// Mitsubishi GX Works2 project: PROJECT55   PLC: FX3G

// global labels: Global1
VAR_GLOBAL
  AnalogOutPut AT D8282 : INT;
  PacketReg AT D1100 : REAL;
  ChocolateToday AT D1102 : REAL;
  TotalChocolate AT D1110 : REAL;
  NutsToday AT D1104 : REAL;
  TotalNuts AT D1112 : REAL;
  FistokToday AT D1106 : REAL;
  TotalFistok AT D1114 : REAL;
  KadaifToday AT D1108 : REAL;
  TotalKadaif AT D1116 : REAL;
  InsertedValue AT M1 : BOOL;
  DayStarted AT M2 : BOOL;
  OutOfStock AT M3 : BOOL;
  DayEnded AT M4 : BOOL;
  EndDay AT X005 : BOOL;
  StartDay AT X007 : BOOL;
  WorkingLight AT Y007 : BOOL;
  MeltingStart AT X001 : BOOL;
END_VAR
VAR_GLOBAL CONSTANT
  MinChocolate : REAL := 400;
  MinNuts : REAL := 100;
  MinFistok : REAL := 120;
  MinKadaif : REAL := 60;
END_VAR
VAR_GLOBAL
  MeltingTank AT D1118 : REAL;
  TransferDone AT M7 : BOOL;
  Sense45 AT X002 : BOOL;
  MeltingLight AT Y001 : BOOL;
  MeltingDone AT M8 : BOOL;
  StockFinished AT M19 : BOOL;
  Sens4Molds AT X003 : BOOL;
  Molds AT D1120 : REAL;
  MoldsTransfer AT M9 : BOOL;
  InMolding AT TC1 : BOOL;
  MoldingFinished AT TS1 : BOOL;
  DuringMolding AT Y002 : BOOL;
END_VAR
VAR_GLOBAL CONSTANT
  MoldingTimee : INT := 40;
END_VAR
VAR_GLOBAL
  Sampling AT X004 : BOOL;
  AnalogInput1 AT D8280 : INT;
  ConvertAnalog AT D1200 : REAL;
END_VAR
VAR_GLOBAL CONSTANT
  ConertNum : REAL := 400;
END_VAR
VAR_GLOBAL
  UserChoice AT D1122 : REAL;
END_VAR
VAR_GLOBAL CONSTANT
  Min5 : REAL := 5;
END_VAR
VAR_GLOBAL
  MakeMixNuts AT M10 : BOOL;
  MakeDubai AT M11 : BOOL;
END_VAR
VAR_GLOBAL CONSTANT
  Count100 : REAL := 100;
END_VAR
VAR_GLOBAL
  MixNutsIngridiants AT M12 : BOOL;
END_VAR
VAR_GLOBAL CONSTANT
  Constant20 : REAL := 2;
  Constant120 : REAL := 2;
  Constant60 : REAL := 60;
END_VAR
VAR_GLOBAL
  DubaiIngridiants AT M13 : BOOL;
END_VAR
VAR_GLOBAL CONSTANT
  Constant100 : REAL := 1;
END_VAR
VAR_GLOBAL
  FillingTank AT D1124 : REAL;
  FillingMixNuts AT M14 : BOOL;
  FillingDubai AT M15 : BOOL;
  FillingDone AT M16 : BOOL;
  Blink AT M0 : BOOL;
  Blink3 AT TC2 : BOOL;
END_VAR
VAR_GLOBAL CONSTANT
  Constant5 : WORD := 5;
END_VAR
VAR_GLOBAL
  StopLight3 AT TS2 : BOOL;
  FillingLight1 AT Y003 : BOOL;
  Blink4 AT TC3 : BOOL;
  StopLight4 AT TS3 : BOOL;
  FillingLight2 AT Y004 : BOOL;
  BlinkingTimer AT TS4 : BOOL;
  StopBlinkingTimer AT TS4 : BOOL;
END_VAR
VAR_GLOBAL CONSTANT
  BlinkingTime : WORD := 50;
END_VAR
VAR_GLOBAL
  Cooling AT X006 : BOOL;
  CoolingTank AT D1126 : REAL;
  CoolingTransfer AT M17 : BOOL;
  CoolingTimer AT TC5 : BOOL;
  StopCoolingTimer AT TS5 : BOOL;
  CoolingLight AT Y006 : BOOL;
END_VAR
VAR_GLOBAL CONSTANT
  CoolingTime : INT := 30;
END_VAR
VAR_GLOBAL
  PackingMachine AT D1128 : REAL;
  PackingTransfer AT M18 : BOOL;
END_VAR
VAR_GLOBAL CONSTANT
  Packing : WORD := 4;
END_VAR
VAR_GLOBAL
  OnePack AT X000 : BOOL;
  PacketsCounter AT CC1 : BOOL;
  StopPacketsCounter AT CS1 : BOOL;
  PackingLight AT Y005 : BOOL;
END_VAR
VAR_GLOBAL CONSTANT
  Constant1 : REAL := 1;
  Constant40 : REAL := 40;
END_VAR
VAR_GLOBAL
  DailyPackets AT D1130 : REAL;
  Cooling1 AT M30 : BOOL;
END_VAR
VAR_GLOBAL CONSTANT
  Min6 : REAL := 6;
  Count20 : REAL := 20;
  Count120 : REAL := 120;
  Count60 : REAL := 60;
  Constant01 : WORD := 1;
END_VAR
VAR_GLOBAL
  PacketsRegg AT TS6 : BOOL;
  EndIteration AT M20 : BOOL;
  PacketsReg AT TS6 : BOOL;
END_VAR

// task Task_01 (event TRUE, interval 0, priority 31): POU_01

PROGRAM POU_01
(* structured ladder/FBD written out as ST: instructions are called as NAME(EN, inputs, outputs); _pN, _eN, _tN stand for wires *)
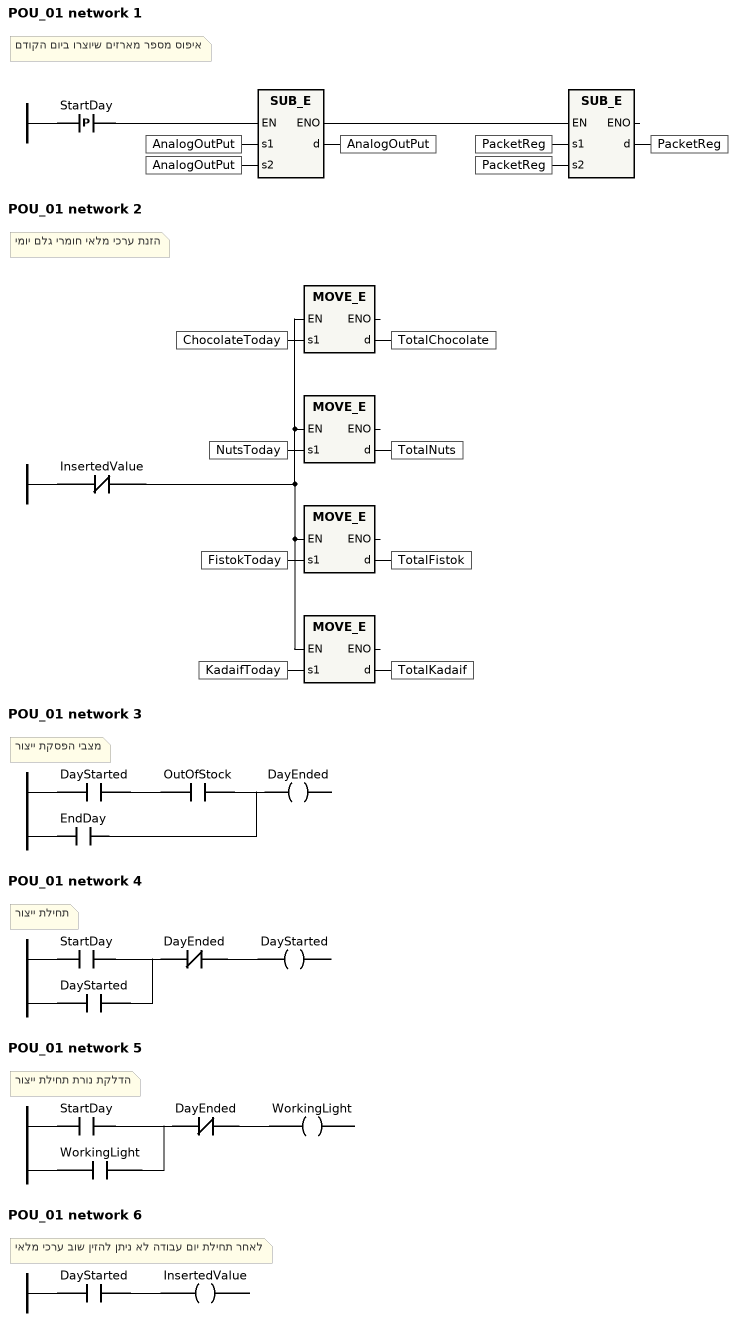
(* network 1 *)
(* איפוס מספר מארזים שיוצרו ביום הקודם *)
_e1 := SUB_E(LDP(TRUE, StartDay), AnalogOutPut, AnalogOutPut, AnalogOutPut);
SUB_E(_e1, PacketReg, PacketReg, PacketReg);
(* network 2 *)
(* הזנת ערכי מלאי חומרי גלם יומי *)
_p1 := NOT InsertedValue;
MOVE_E(_p1, ChocolateToday, TotalChocolate);
MOVE_E(_p1, NutsToday, TotalNuts);
MOVE_E(_p1, FistokToday, TotalFistok);
MOVE_E(_p1, KadaifToday, TotalKadaif);
(* network 3 *)
(* מצבי הפסקת ייצור *)
DayEnded := (DayStarted AND OutOfStock) OR EndDay;
(* network 4 *)
(* תחילת ייצור *)
DayStarted := (StartDay OR DayStarted) AND NOT DayEnded;
(* network 5 *)
(* הדלקת נורת תחילת ייצור *)
WorkingLight := (StartDay OR WorkingLight) AND NOT DayEnded;
(* network 6 *)
(* לאחר תחילת יום עבודה לא ניתן להזין שוב ערכי מלאי *)
InsertedValue := DayStarted;
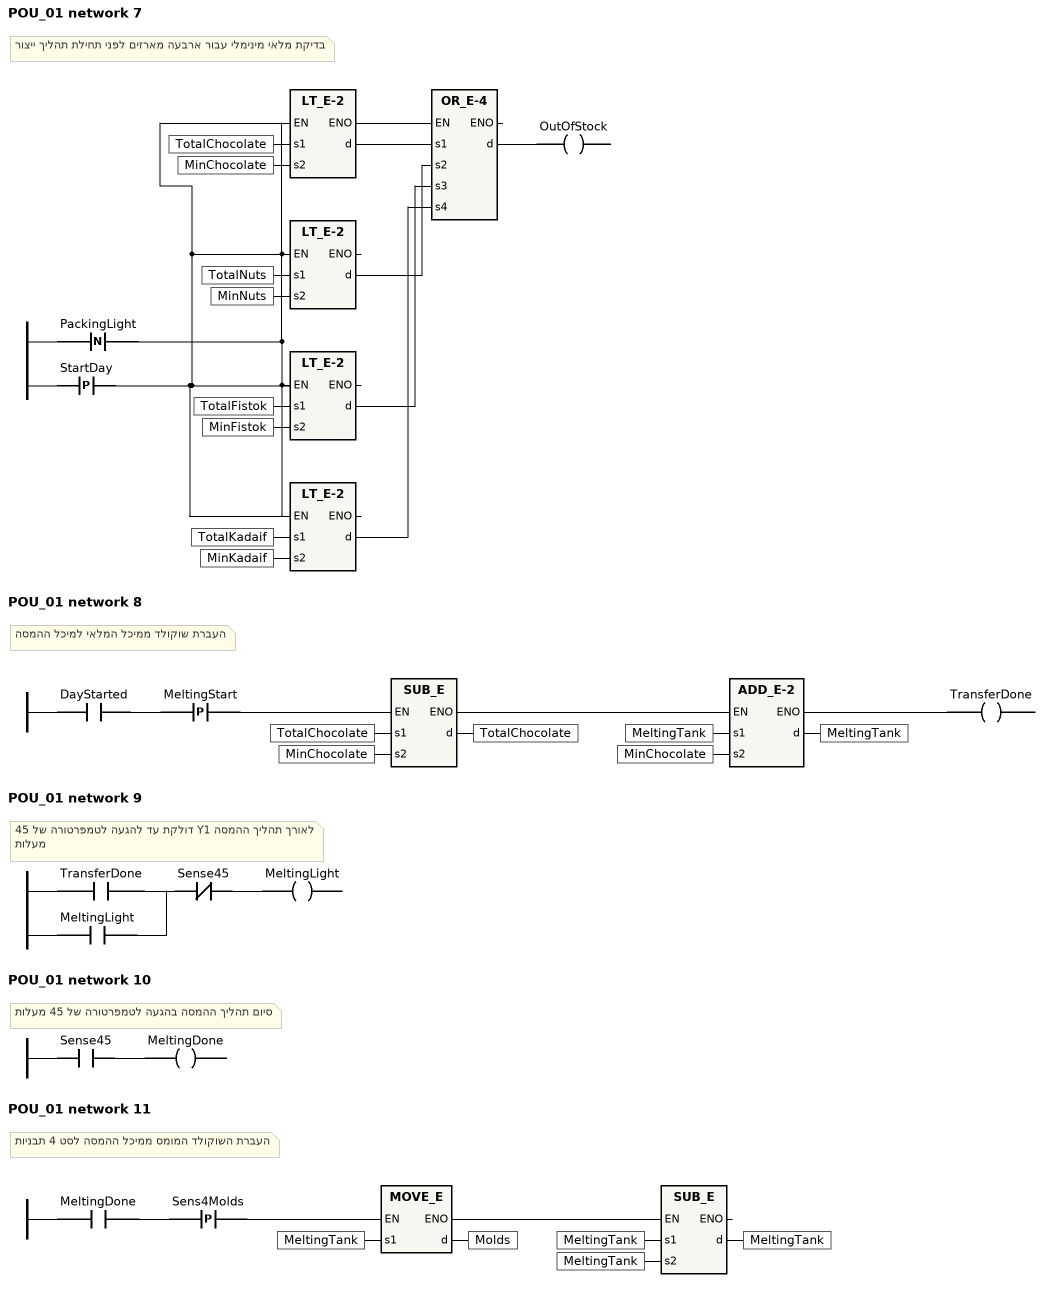
(* network 7 *)
(* בדיקת מלאי מינימלי עבור ארבעה מארזים לפני תחילת תהליך ייצור *)
_p1 := LDF(TRUE, PackingLight) OR LDP(TRUE, StartDay);
_e3 := LT_E(_p1, TotalChocolate, MinChocolate, _t2);
LT_E(_p1, TotalNuts, MinNuts, _t4);
LT_E(_p1, TotalFistok, MinFistok, _t5);
LT_E(_p1, TotalKadaif, MinKadaif, _t6);
OR_E(_e3, _t2, _t4, _t5, _t6, _t7);
OutOfStock := _t7;
(* network 8 *)
(* העברת שוקולד ממיכל המלאי למיכל ההמסה *)
_e1 := SUB_E(DayStarted AND LDP(TRUE, MeltingStart), TotalChocolate, MinChocolate, TotalChocolate);
_e2 := ADD_E(_e1, MeltingTank, MinChocolate, MeltingTank);
TransferDone := _e2;
(* network 9 *)
(* לאורך תהליך ההמסה Y1 דולקת עד להגעה לטמפרטורה של 45 מעלות *)
MeltingLight := (TransferDone OR MeltingLight) AND NOT Sense45;
(* network 10 *)
(* סיום תהליך ההמסה בהגעה לטמפרטורה של 45 מעלות *)
MeltingDone := Sense45;
(* network 11 *)
(* העברת השוקולד המומס ממיכל ההמסה לסט 4 תבניות *)
_e1 := MOVE_E(MeltingDone AND LDP(TRUE, Sens4Molds), MeltingTank, Molds);
SUB_E(_e1, MeltingTank, MeltingTank, MeltingTank);
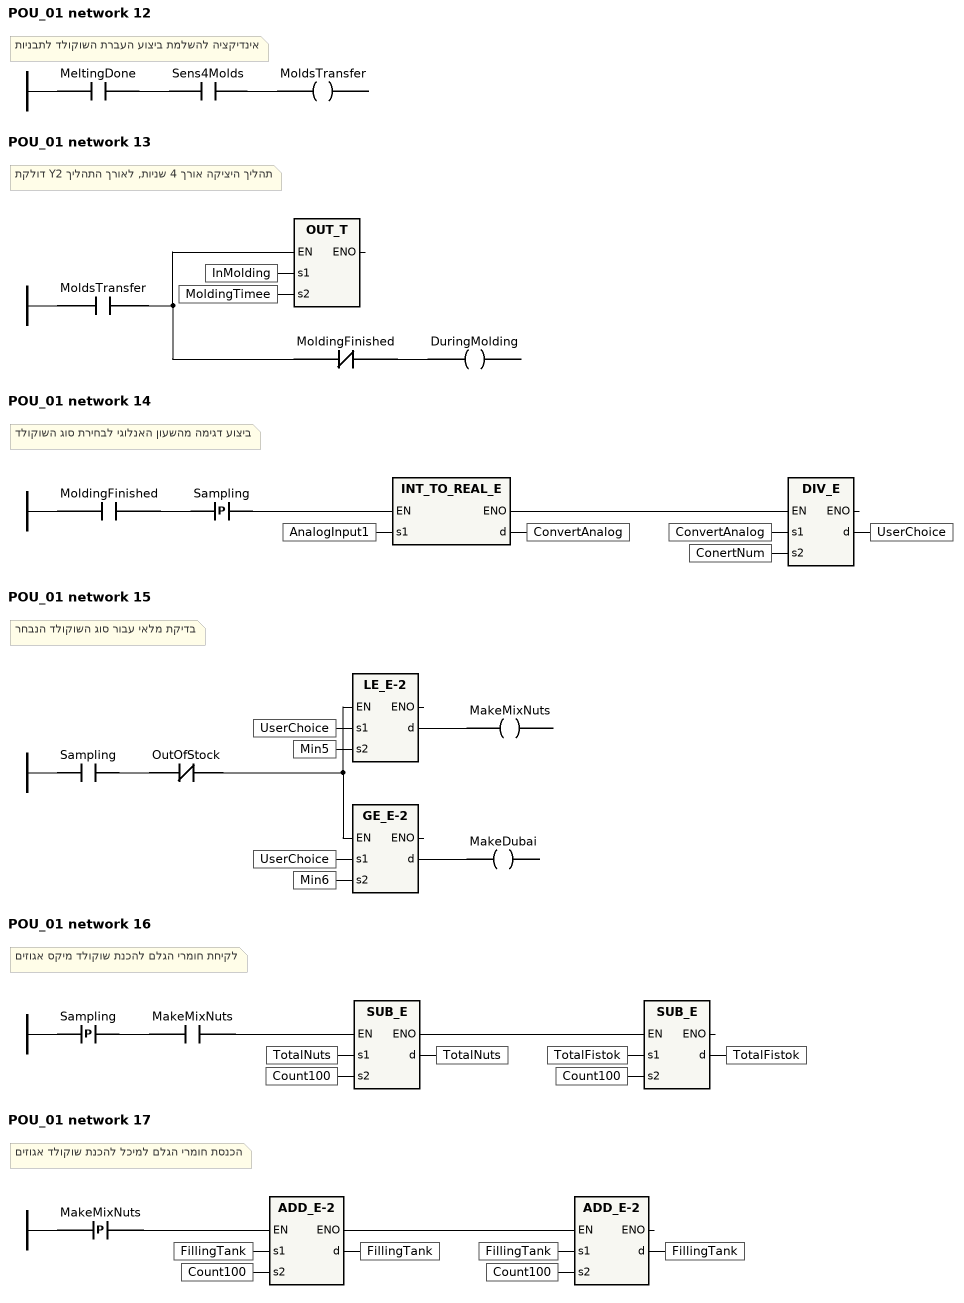
(* network 12 *)
(* אינדיקציה להשלמת ביצוע העברת השוקולד לתבניות *)
MoldsTransfer := MeltingDone AND Sens4Molds;
(* network 13 *)
(* תהליך היציקה אורך 4 שניות, לאורך התהליך Y2 דולקת *)
OUT_T(MoldsTransfer, InMolding, MoldingTimee);
DuringMolding := MoldsTransfer AND NOT MoldingFinished;
(* network 14 *)
(* ביצוע דגימה מהשעון האנלוגי לבחירת סוג השוקולד *)
_e1 := INT_TO_REAL_E(MoldingFinished AND LDP(TRUE, Sampling), AnalogInput1, ConvertAnalog);
DIV_E(_e1, ConvertAnalog, ConertNum, UserChoice);
(* network 15 *)
(* בדיקת מלאי עבור סוג השוקולד הנבחר *)
_p1 := Sampling AND NOT OutOfStock;
LE_E(_p1, UserChoice, Min5, _t2);
MakeMixNuts := _t2;
GE_E(_p1, UserChoice, Min6, _t3);
MakeDubai := _t3;
(* network 16 *)
(* לקיחת חומרי הגלם להכנת שוקולד מיקס אגוזים *)
_e1 := SUB_E(LDP(TRUE, Sampling) AND MakeMixNuts, TotalNuts, Count100, TotalNuts);
SUB_E(_e1, TotalFistok, Count100, TotalFistok);
(* network 17 *)
(* הכנסת חומרי הגלם למיכל להכנת שוקולד אגוזים *)
_e1 := ADD_E(LDP(TRUE, MakeMixNuts), FillingTank, Count100, FillingTank);
ADD_E(_e1, FillingTank, Count100, FillingTank);
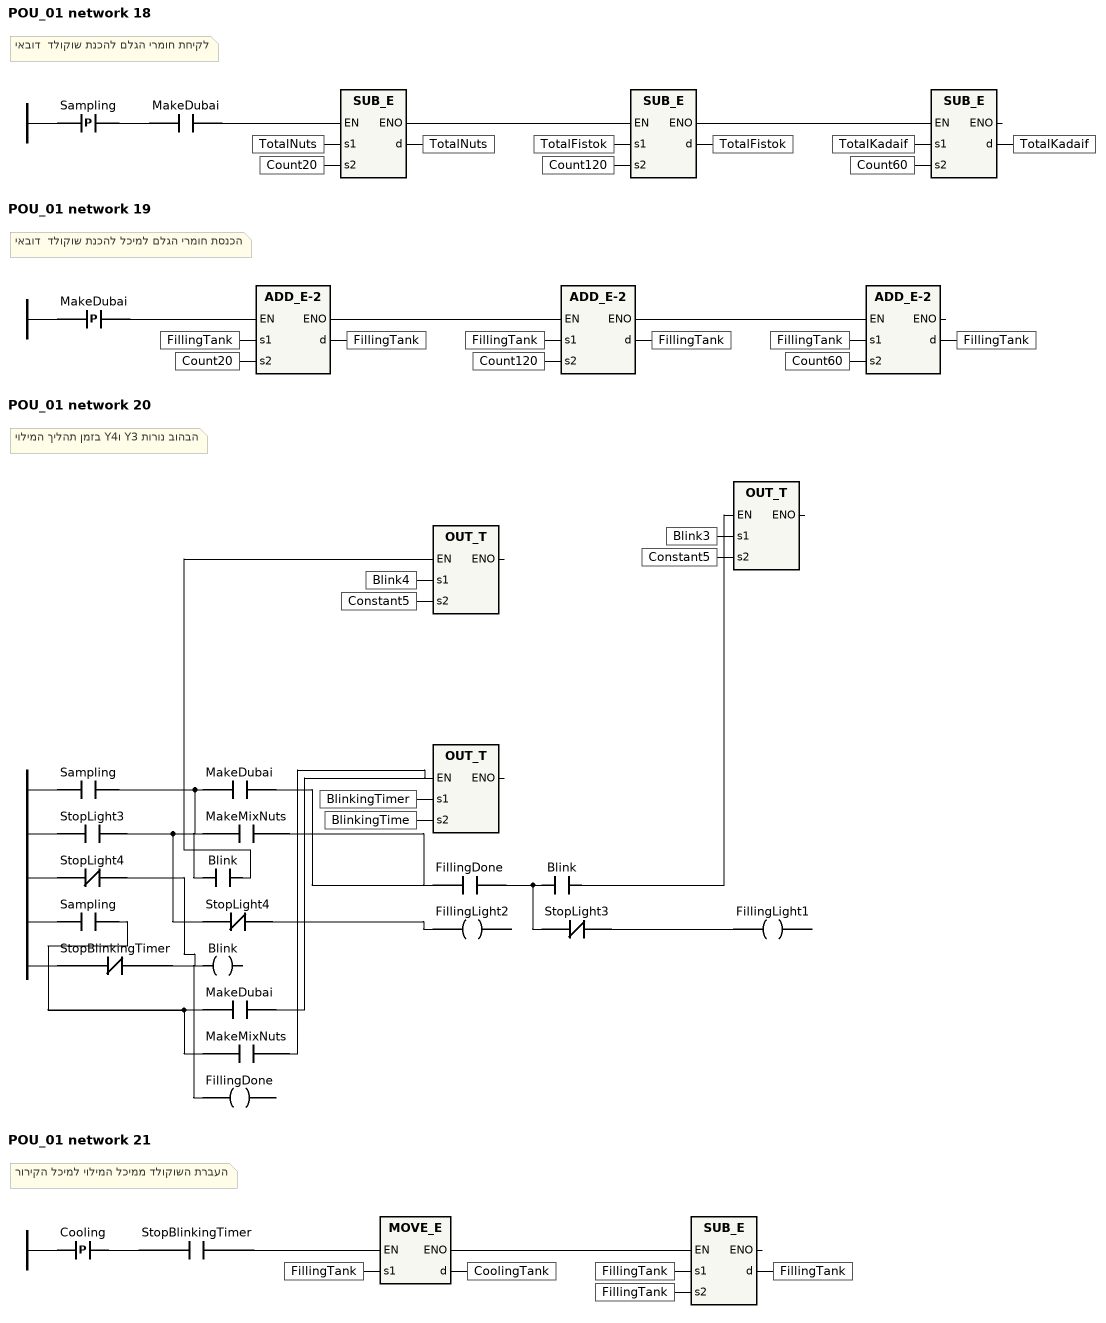
(* network 18 *)
(* לקיחת חומרי הגלם להכנת שוקולד  דובאי *)
_e1 := SUB_E(LDP(TRUE, Sampling) AND MakeDubai, TotalNuts, Count20, TotalNuts);
_e2 := SUB_E(_e1, TotalFistok, Count120, TotalFistok);
SUB_E(_e2, TotalKadaif, Count60, TotalKadaif);
(* network 19 *)
(* הכנסת חומרי הגלם למיכל להכנת שוקולד  דובאי *)
_e1 := ADD_E(LDP(TRUE, MakeDubai), FillingTank, Count20, FillingTank);
_e2 := ADD_E(_e1, FillingTank, Count120, FillingTank);
ADD_E(_e2, FillingTank, Count60, FillingTank);
(* network 20 *)
(* הבהוב נורות Y3 וY4 בזמן תהליך המילוי *)
_p1 := ((Sampling AND MakeDubai) OR (Sampling AND MakeMixNuts)) AND FillingDone;
OUT_T(_p1 AND Blink, Blink3, Constant5);
FillingLight1 := _p1 AND NOT StopLight3;
OUT_T(StopLight3 AND Blink, Blink4, Constant5);
FillingLight2 := StopLight3 AND NOT StopLight4;
Blink := NOT StopLight4;
OUT_T((Sampling AND MakeDubai) OR (Sampling AND MakeMixNuts), BlinkingTimer, BlinkingTime);
FillingDone := NOT StopBlinkingTimer;
(* network 21 *)
(* העברת השוקולד ממיכל המילוי למיכל הקירור *)
_e1 := MOVE_E(LDP(TRUE, Cooling) AND StopBlinkingTimer, FillingTank, CoolingTank);
SUB_E(_e1, FillingTank, FillingTank, FillingTank);
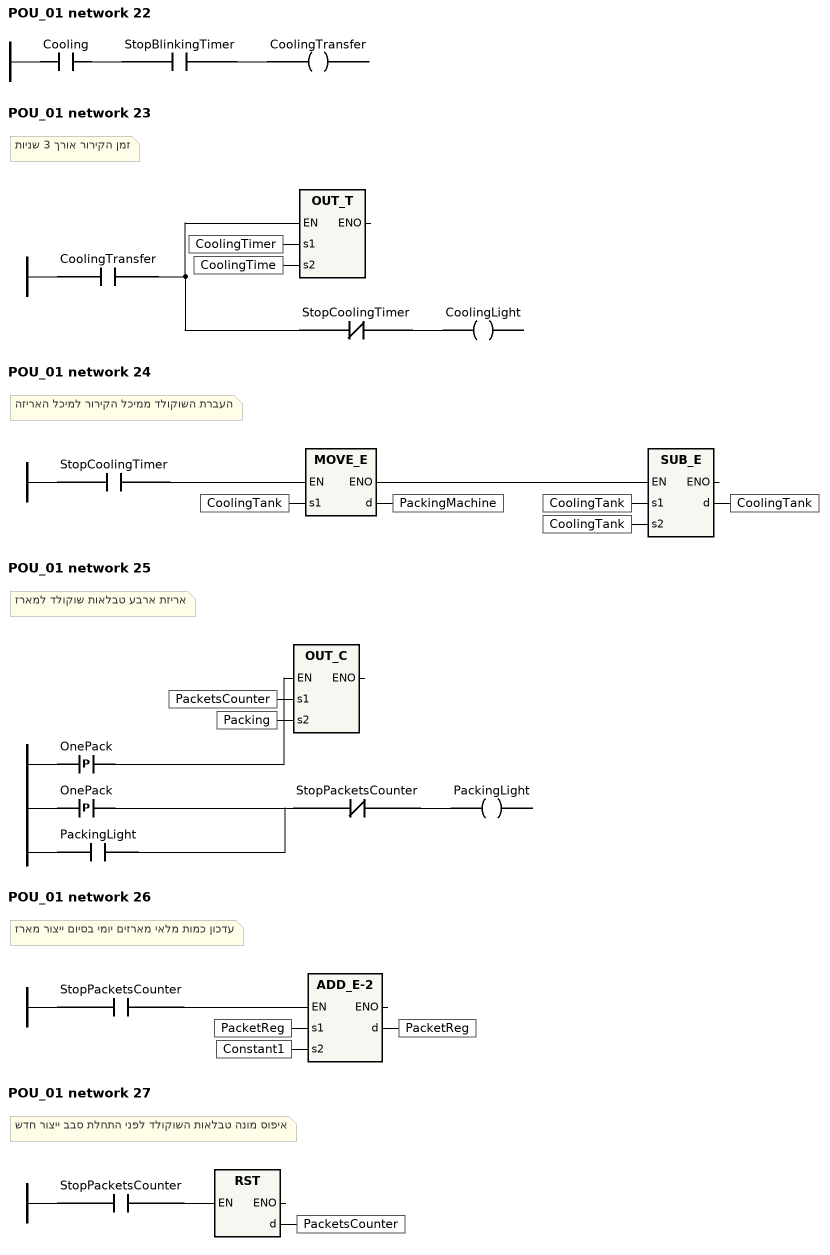
(* network 22 *)
CoolingTransfer := Cooling AND StopBlinkingTimer;
(* network 23 *)
(* זמן הקירור אורך 3 שניות *)
OUT_T(CoolingTransfer, CoolingTimer, CoolingTime);
CoolingLight := CoolingTransfer AND NOT StopCoolingTimer;
(* network 24 *)
(* העברת השוקולד ממיכל הקירור למיכל האריזה *)
_e1 := MOVE_E(StopCoolingTimer, CoolingTank, PackingMachine);
SUB_E(_e1, CoolingTank, CoolingTank, CoolingTank);
(* network 25 *)
(* אריזת ארבע טבלאות שוקולד למארז *)
OUT_C(LDP(TRUE, OnePack), PacketsCounter, Packing);
PackingLight := (LDP(TRUE, OnePack) OR PackingLight) AND NOT StopPacketsCounter;
(* network 26 *)
(* עדכון כמות מלאי מארזים יומי בסיום ייצור מארז *)
ADD_E(StopPacketsCounter, PacketReg, Constant1, PacketReg);
(* network 27 *)
(* איפוס מונה טבלאות השוקולד לפני התחלת סבב ייצור חדש *)
RST(StopPacketsCounter, PacketsCounter);
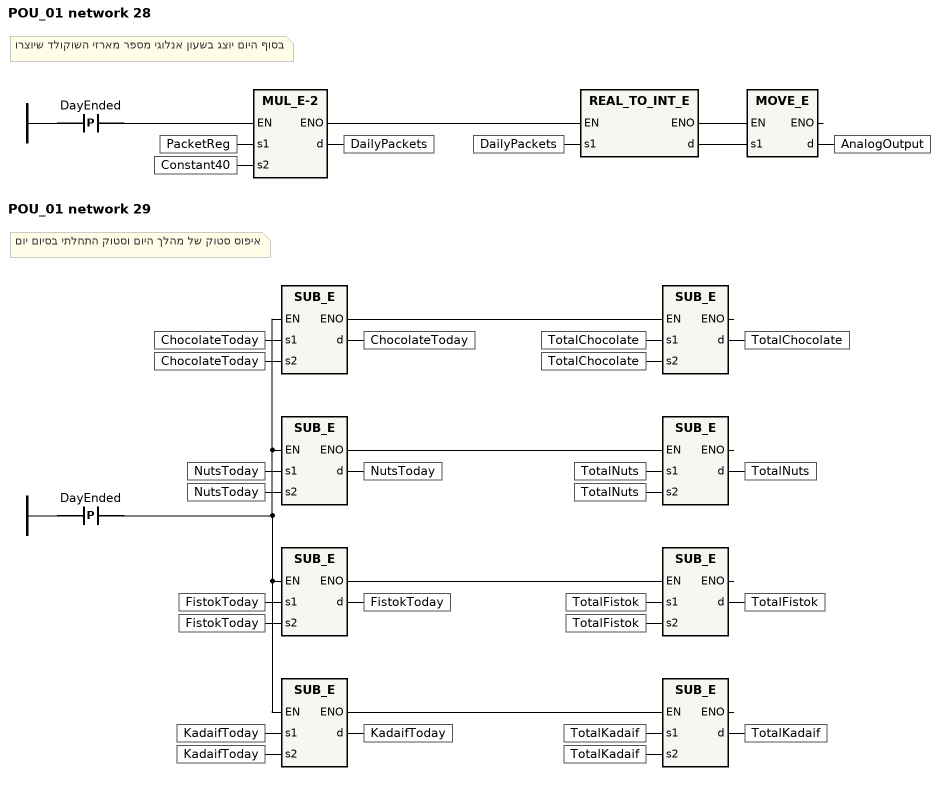
(* network 28 *)
(* בסוף היום יוצג בשעון אנלוגי מספר מארזי השוקולד שיוצרו *)
_e1 := MUL_E(LDP(TRUE, DayEnded), PacketReg, Constant40, DailyPackets);
_e3 := REAL_TO_INT_E(_e1, DailyPackets, _t2);
MOVE_E(_e3, _t2, AnalogOutput);
(* network 29 *)
(* איפוס סטוק של מהלך היום וסטוק התחלתי בסיום יום *)
_p1 := LDP(TRUE, DayEnded);
_e2 := SUB_E(_p1, ChocolateToday, ChocolateToday, ChocolateToday);
SUB_E(_e2, TotalChocolate, TotalChocolate, TotalChocolate);
_e3 := SUB_E(_p1, NutsToday, NutsToday, NutsToday);
SUB_E(_e3, TotalNuts, TotalNuts, TotalNuts);
_e4 := SUB_E(_p1, FistokToday, FistokToday, FistokToday);
SUB_E(_e4, TotalFistok, TotalFistok, TotalFistok);
_e5 := SUB_E(_p1, KadaifToday, KadaifToday, KadaifToday);
SUB_E(_e5, TotalKadaif, TotalKadaif, TotalKadaif);
END_PROGRAM
